# EPICS substitutions: mpgSupport/Db/ioc/edefSim.substitutions
# one per system - declare EVG stuff in this IOC for testing

file mpgEventAll.db
{
#                               Check    Trigger
#          Device             PNET Data  Seq Ram
  pattern { DEVICE     , SYSI , CHECKI , SENDI }
          { IOC:SYS1:1 , SYS1 ,   0    ,   0   }
}
file bsaEdefAll.db {
  pattern { DEVICE     , SYSI }
 	  { IOC:SYS1:1 , SYS1 }
}
file evrPatternAll.db {
#	    Device     , Time Slot Processing      PNET Processing  BSA Data Processing
  pattern { DEVICE     ,         LINK4          ,      LINK5      ,      LINK6        }
	  { IOC:SYS1:1 , IOC:SYS1:1:TIMESLOTN-1 , IOC:SYS1:1:PNET , IOC:SYS1:1:EDEFFO }
}
file mpgPatternTest.db {
  pattern { SYSI  , UNITI }
 	  { SYS1  ,  1    }
}
